FUNCTION_BLOCK Demo2 (* HMI Panel Type *)
  (* Standard: 61499-2 *)
  (* Version 0.1, 2014-08-21, WD, YY Automation *)
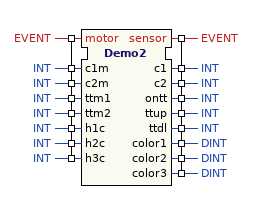
  EVENT_INPUT
    motor : EVENT WITH c1m, c2m, ttm1, ttm2, h1c, h2c, h3c; (* Service Initialization *)
  END_EVENT
  EVENT_OUTPUT
    sensor : EVENT WITH c1, c2, ontt, ttup, ttdl, color1, color2, color3; (* Initialization Confirm *)
  END_EVENT
  VAR_INPUT
    c1m : INT;
    c2m : INT;
    ttm1 : INT;
    ttm2 : INT;
    h1c : INT;
    h2c : INT;
    h3c : INT;
  END_VAR
  VAR_OUTPUT
    c1 : INT; (* Event Output Qualifier *)
    c2 : INT;
    ontt : INT;
    ttup : INT;
    ttdl : INT;
    color1 : DINT;
    color2 : DINT;
    color3 : DINT;
  END_VAR
END_FUNCTION_BLOCK
(* other elements stored in the file *)
(* Panel Language=HTML Width=1200 Height=1000 *)
(* PanelHTML  <div ng-controller="<%id%>Controller" style="position: absolute; top: <%top%>px; left: <%left%>px; width: <%width%>px; height: <%height%>px; background: <%background%>;"> <div data-ng-init="connect()"></div> </div> *)
